// TIA Portal project "Kemence" (V15.1)

(* hardware
DEVICE "HMI_1"  KTP600 Basic color PN
   slot 0: "HMI_1"  KTP600 Basic color PN  6AV6 647-0AD11-3AX0  12.0.0.0
   slot 1: "HMI_RT_1"  KTP600 Basic color PN  6AV6 647-0AD11-3AX0  12.0.0.0
   slot 5: "HMI_1.IE_CP_1"  PROFINET Interface  12.0.0.0
      slot 1: "PROFINET Interface_1"  PROFINET Interface
         slot 1: "Port_1"  Port
DEVICE "S7300/ET200M station_2"  S7-300 station
   slot 0: "Rail_0"  Rail  6ES7 390-1***0-0AA0
   slot 2: "PLC_2"  CPU 314C-2 PN/DP  6ES7 314-6EH04-0AB0  V3.3
      slot 2: "PROFINET interface_1"  PN-IO
         slot 1: "Port_1"  Port
         slot 2: "Port_2"  Port
      slot 5: "DI 24/DO 16_1"  DI24/DO16
      slot 6: "AI 5/AO 2_1"  AI5/AO2
      slot 7: "Count_1"  Counter
      slot 8: "Positioning_1"  Positioning
*)

// ===== PLC "PLC_2"  CPU 314C-2 PN/DP =====

VAR_GLOBAL   // PLC tag table "Default tag table"
   "Homerseklet" AT %IW808 : Int;
   "Ki" AT %Q136.0 : Bool;
   "Orajel" AT %M0.5 : Bool;
END_VAR

DATA_BLOCK "Valtozoim"   // DB1
{ S7_Optimized_Access := 'FALSE' }
VERSION : 0.1
   VAR
      Aktualis : Int;
      Eloirt : Int;
      Hiszterezis : Int;
      Start1 : Bool;
      Start2 : Bool;
      Start3 : Bool;
      "On/Off" : Bool;
      Eloirt_plusz_Hister : Int;
      Eloirt_minus_Hister : Int;
      Kimenet : Bool;
      Komment : Bool;
      Error : Int;
      U : Int;
      Kp : Int;
      Pulse : Bool := true;
   END_VAR
BEGIN
END_DATA_BLOCK

DATA_BLOCK "Harmadik_pont"   // DB5
{ S7_Optimized_Access := 'FALSE' }
VERSION : 0.1
   VAR
      Man_on : Bool;
      PID : Bool;
      CYKLE_TIME : Time;
      Eloirt_REAL : Real;
      Aktualis_REAL : Real;
      Kp_REAL : Real;
      Integralasi_periodus : Time;
      Derivalasi_periodus : Time;
      Felso_hatar : Real;
      Also_hatar : Real;
      szabalyzo_jel : Real;
      Aktualis_DINT : DInt;
      Eloirt_DINT : DInt;
      KP_REAL_1 : Real;
      U_DINT : DInt;
      U_INT : Int;
   END_VAR
BEGIN
END_DATA_BLOCK

FUNCTION "Block_2" : Void   // FC1, LAD
{ S7_Optimized_Access := 'FALSE' }
VERSION : 0.1
BEGIN

REGION Network 1
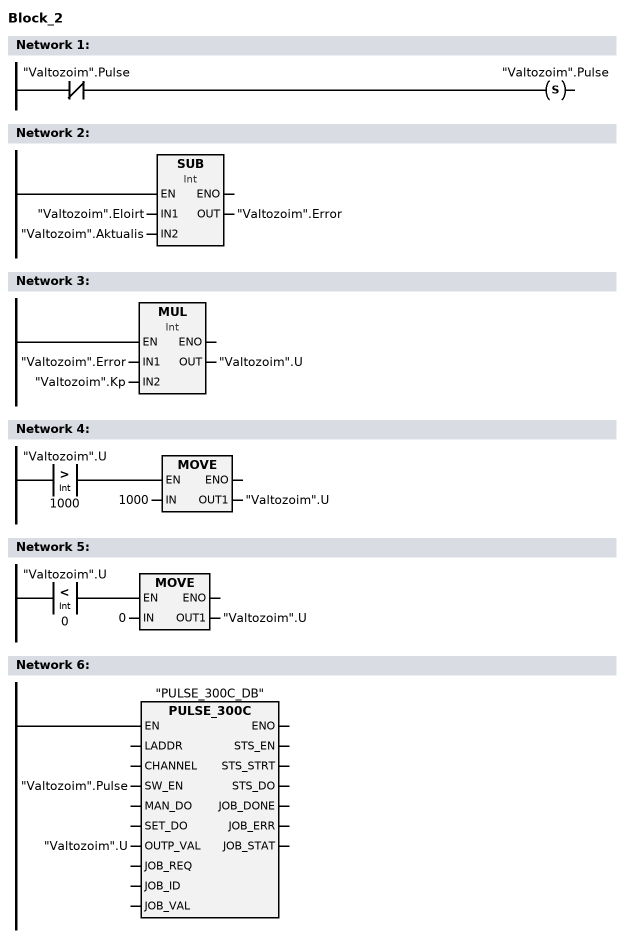
   RUNG wire#powerrail
      I_Contact( "Valtozoim".Pulse )
      S_Coil( "Valtozoim".Pulse )
   END_RUNG
   // the same network as SCL:
   IF NOT "Valtozoim".Pulse THEN "Valtozoim".Pulse := TRUE; END_IF;
END_REGION

REGION Network 2
   RUNG wire#powerrail
      { S7_Templates := "SrcType := Int"; S7_GenerateENO := "TRUE" } Sub(in1 := "Valtozoim".Eloirt, in2 := "Valtozoim".Aktualis, out => "Valtozoim".Error)
   END_RUNG
   // the same network as SCL:
   "Valtozoim".Error := "Valtozoim".Eloirt - "Valtozoim".Aktualis;
END_REGION

REGION Network 3
   RUNG wire#powerrail
      { S7_Templates := "SrcType := Int"; S7_GenerateENO := "TRUE" } Mul(in1 := "Valtozoim".Error, in2 := "Valtozoim".Kp, out => "Valtozoim".U)
   END_RUNG
   // the same network as SCL:
   "Valtozoim".U := "Valtozoim".Error * "Valtozoim".Kp;
END_REGION

REGION Network 4
   RUNG wire#powerrail
      { S7_Templates := "SrcType := Int" } GT_Contact(in1 := "Valtozoim".U, in2 := 1000)
      { S7_GenerateENO := "TRUE" } Move(in := 1000, out1 => "Valtozoim".U)
   END_RUNG
   // the same network as SCL:
   IF "Valtozoim".U > 1000 THEN "Valtozoim".U := 1000; END_IF;
END_REGION

REGION Network 5
   RUNG wire#powerrail
      { S7_Templates := "SrcType := Int" } LT_Contact(in1 := "Valtozoim".U, in2 := 0)
      { S7_GenerateENO := "TRUE" } Move(in := 0, out1 => "Valtozoim".U)
   END_RUNG
   // the same network as SCL:
   IF "Valtozoim".U < 0 THEN "Valtozoim".U := 0; END_IF;
END_REGION

REGION Network 6
   "PULSE_300C_DB"(SW_EN := "Valtozoim".Pulse, OUTP_VAL := "Valtozoim".U);   // PULSE_300C
END_REGION
END_FUNCTION

FUNCTION "Block_1" : Void   // FC2, LAD
{ S7_Optimized_Access := 'FALSE' }
VERSION : 0.1
BEGIN

REGION Network 1
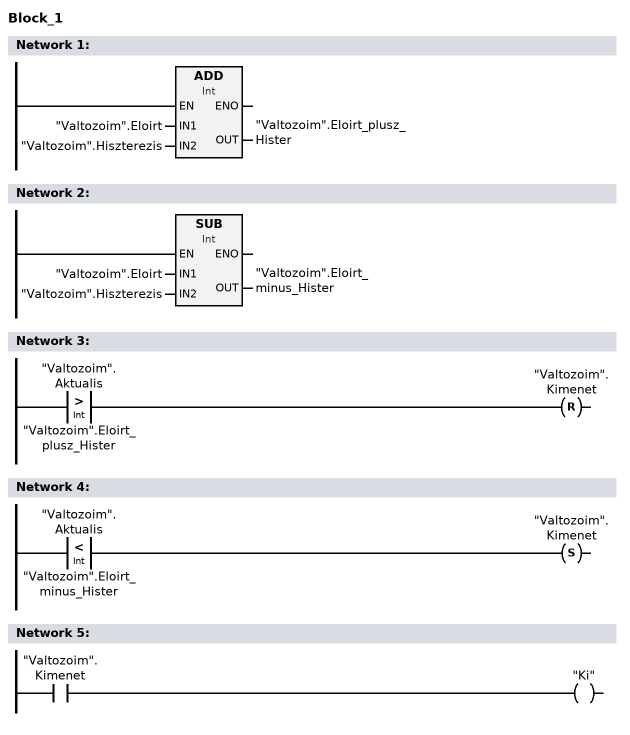
   RUNG wire#powerrail
      { S7_Templates := "SrcType := Int"; S7_GenerateENO := "TRUE" } Add(in1 := "Valtozoim".Eloirt, in2 := "Valtozoim".Hiszterezis, out => "Valtozoim".Eloirt_plusz_Hister)
   END_RUNG
   // the same network as SCL:
   "Valtozoim".Eloirt_plusz_Hister := "Valtozoim".Eloirt + "Valtozoim".Hiszterezis;
END_REGION

REGION Network 2
   RUNG wire#powerrail
      { S7_Templates := "SrcType := Int"; S7_GenerateENO := "TRUE" } Sub(in1 := "Valtozoim".Eloirt, in2 := "Valtozoim".Hiszterezis, out => "Valtozoim".Eloirt_minus_Hister)
   END_RUNG
   // the same network as SCL:
   "Valtozoim".Eloirt_minus_Hister := "Valtozoim".Eloirt - "Valtozoim".Hiszterezis;
END_REGION

REGION Network 3
   RUNG wire#powerrail
      { S7_Templates := "SrcType := Int" } GT_Contact(in1 := "Valtozoim".Aktualis, in2 := "Valtozoim".Eloirt_plusz_Hister)
      R_Coil( "Valtozoim".Kimenet )
   END_RUNG
   // the same network as SCL:
   IF "Valtozoim".Aktualis > "Valtozoim".Eloirt_plusz_Hister THEN "Valtozoim".Kimenet := FALSE; END_IF;
END_REGION

REGION Network 4
   RUNG wire#powerrail
      { S7_Templates := "SrcType := Int" } LT_Contact(in1 := "Valtozoim".Aktualis, in2 := "Valtozoim".Eloirt_minus_Hister)
      S_Coil( "Valtozoim".Kimenet )
   END_RUNG
   // the same network as SCL:
   IF "Valtozoim".Aktualis < "Valtozoim".Eloirt_minus_Hister THEN "Valtozoim".Kimenet := TRUE; END_IF;
END_REGION

REGION Network 5
   RUNG wire#powerrail
      Contact( "Valtozoim".Kimenet )
      Coil( "Ki" )
   END_RUNG
   // the same network as SCL:
   "Ki" := "Valtozoim".Kimenet;
END_REGION
END_FUNCTION

FUNCTION "Block_3" : Void   // FC3, LAD
{ S7_Optimized_Access := 'FALSE' }
VERSION : 0.1
BEGIN

REGION Network 1
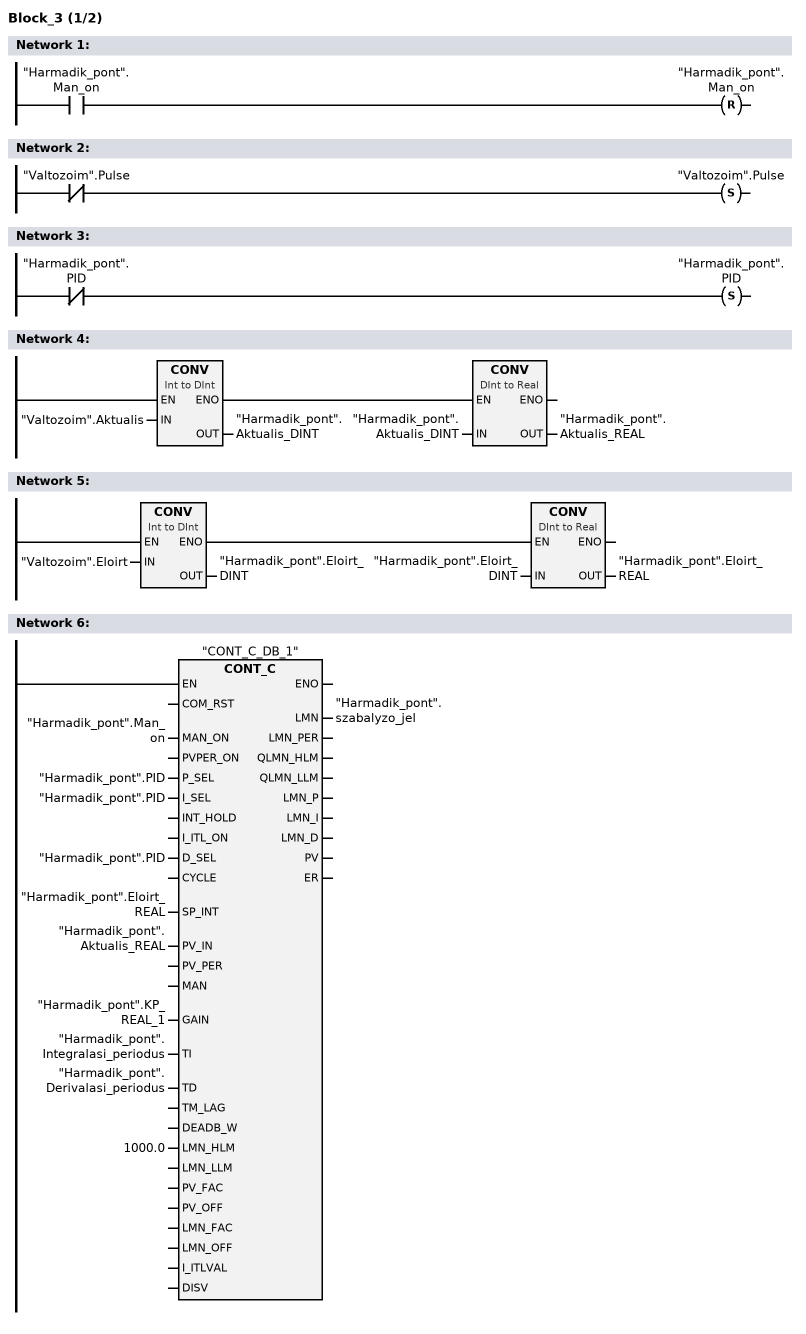
   RUNG wire#powerrail
      Contact( "Harmadik_pont".Man_on )
      R_Coil( "Harmadik_pont".Man_on )
   END_RUNG
   // the same network as SCL:
   IF "Harmadik_pont".Man_on THEN "Harmadik_pont".Man_on := FALSE; END_IF;
END_REGION

REGION Network 2
   RUNG wire#powerrail
      I_Contact( "Valtozoim".Pulse )
      S_Coil( "Valtozoim".Pulse )
   END_RUNG
   // the same network as SCL:
   IF NOT "Valtozoim".Pulse THEN "Valtozoim".Pulse := TRUE; END_IF;
END_REGION

REGION Network 3
   RUNG wire#powerrail
      I_Contact( "Harmadik_pont".PID )
      S_Coil( "Harmadik_pont".PID )
   END_RUNG
   // the same network as SCL:
   IF NOT "Harmadik_pont".PID THEN "Harmadik_pont".PID := TRUE; END_IF;
END_REGION

REGION Network 4
   RUNG wire#powerrail
      { S7_Templates := "[SrcType := Int, DestType := DInt]"; S7_GenerateENO := "TRUE" } Convert(in := "Valtozoim".Aktualis, out => "Harmadik_pont".Aktualis_DINT)
      { S7_Templates := "[SrcType := DInt, DestType := Real]"; S7_GenerateENO := "TRUE" } Convert(in := "Harmadik_pont".Aktualis_DINT, out => "Harmadik_pont".Aktualis_REAL)
   END_RUNG
   // the same network as SCL:
   // ENO of a box is taken as its EN; it also drops when the box reports an error
   "Harmadik_pont".Aktualis_DINT := INT_TO_DINT("Valtozoim".Aktualis);
   "Harmadik_pont".Aktualis_REAL := DINT_TO_REAL("Harmadik_pont".Aktualis_DINT);
END_REGION

REGION Network 5
   RUNG wire#powerrail
      { S7_Templates := "[SrcType := Int, DestType := DInt]"; S7_GenerateENO := "TRUE" } Convert(in := "Valtozoim".Eloirt, out => "Harmadik_pont".Eloirt_DINT)
      { S7_Templates := "[SrcType := DInt, DestType := Real]"; S7_GenerateENO := "TRUE" } Convert(in := "Harmadik_pont".Eloirt_DINT, out => "Harmadik_pont".Eloirt_REAL)
   END_RUNG
   // the same network as SCL:
   // ENO of a box is taken as its EN; it also drops when the box reports an error
   "Harmadik_pont".Eloirt_DINT := INT_TO_DINT("Valtozoim".Eloirt);
   "Harmadik_pont".Eloirt_REAL := DINT_TO_REAL("Harmadik_pont".Eloirt_DINT);
END_REGION

REGION Network 6
   "CONT_C_DB_1"(MAN_ON := "Harmadik_pont".Man_on,   // CONT_C
                 P_SEL := "Harmadik_pont".PID,
                 I_SEL := "Harmadik_pont".PID,
                 D_SEL := "Harmadik_pont".PID,
                 SP_INT := "Harmadik_pont".Eloirt_REAL,
                 PV_IN := "Harmadik_pont".Aktualis_REAL,
                 GAIN := "Harmadik_pont".KP_REAL_1,
                 TI := "Harmadik_pont".Integralasi_periodus,
                 TD := "Harmadik_pont".Derivalasi_periodus,
                 LMN_HLM := 1000.0,
                 LMN => "Harmadik_pont".szabalyzo_jel);
END_REGION

REGION Network 7
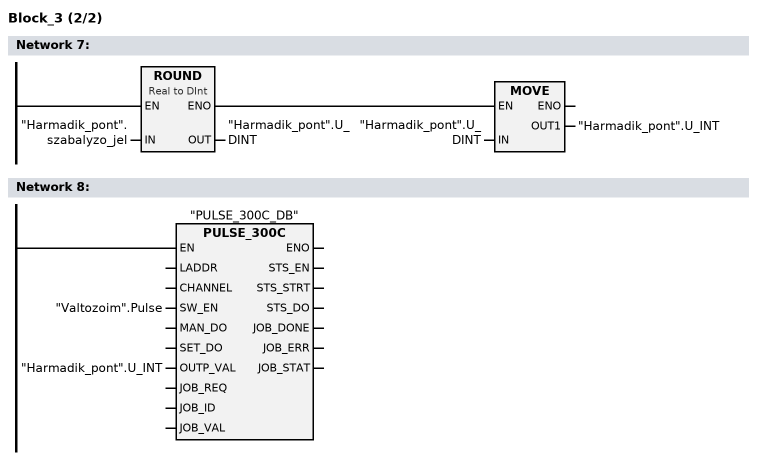
   RUNG wire#powerrail
      { S7_Templates := "[SrcType := Real, DestType := DInt]"; S7_GenerateENO := "TRUE" } Round(in := "Harmadik_pont".szabalyzo_jel, out => "Harmadik_pont".U_DINT)
      { S7_GenerateENO := "TRUE" } Move(in := "Harmadik_pont".U_DINT, out1 => "Harmadik_pont".U_INT)
   END_RUNG
   // the same network as SCL:
   // ENO of a box is taken as its EN; it also drops when the box reports an error
   "Harmadik_pont".U_DINT := ROUND("Harmadik_pont".szabalyzo_jel);
   "Harmadik_pont".U_INT := "Harmadik_pont".U_DINT;
END_REGION

REGION Network 8
   "PULSE_300C_DB"(SW_EN := "Valtozoim".Pulse, OUTP_VAL := "Harmadik_pont".U_INT);   // PULSE_300C
END_REGION
END_FUNCTION

ORGANIZATION_BLOCK "Main"   // OB1, LAD
TITLE = "Main Program Sweep (Cycle)"
{ S7_Optimized_Access := 'FALSE' }
VERSION : 0.1
   VAR_TEMP
      OB1_EV_CLASS : Byte;   // Bits 0-3 = 1 (Coming event), Bits 4-7 = 1 (Event class 1)
      OB1_SCAN_1 : Byte;   // 1 (Cold restart scan 1 of OB 1), 3 (Scan 2-n of OB 1)
      OB1_PRIORITY : Byte;   // Priority of OB Execution
      OB1_OB_NUMBR : Byte;   // 1 (Organization block 1, OB1)
      OB1_RESERVED_1 : Byte;   // Reserved for system
      OB1_RESERVED_2 : Byte;   // Reserved for system
      OB1_PREV_CYCLE : Int;   // Cycle time of previous OB1 scan (milliseconds)
      OB1_MIN_CYCLE : Int;   // Minimum cycle time of OB1 (milliseconds)
      OB1_MAX_CYCLE : Int;   // Maximum cycle time of OB1 (milliseconds)
      OB1_DATE_TIME : Date_And_Time;   // Date and time OB1 started
   END_VAR
BEGIN

REGION Network 1
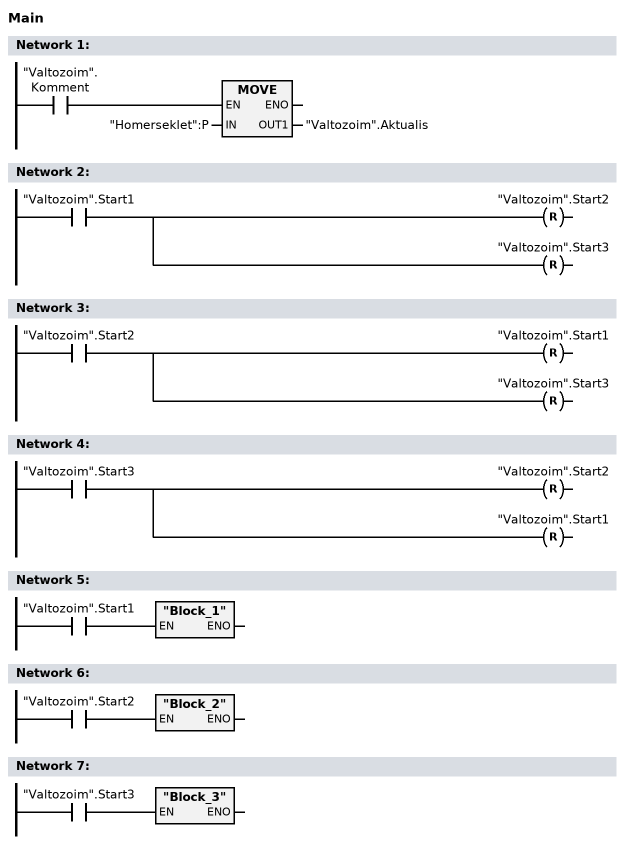
   RUNG wire#powerrail
      Contact( "Valtozoim".Komment )
      { S7_GenerateENO := "TRUE" } Move(in := "Homerseklet":P, out1 => "Valtozoim".Aktualis)
   END_RUNG
   // the same network as SCL:
   IF "Valtozoim".Komment THEN "Valtozoim".Aktualis := "Homerseklet":P; END_IF;
END_REGION

REGION Network 2
   RUNG wire#powerrail
      Contact( "Valtozoim".Start1 )
      wire#w1
      R_Coil( "Valtozoim".Start2 )
   END_RUNG
   RUNG wire#w1
      R_Coil( "Valtozoim".Start3 )
   END_RUNG
   // the same network as SCL:
   IF "Valtozoim".Start1 THEN
       "Valtozoim".Start2 := FALSE;
       "Valtozoim".Start3 := FALSE;
   END_IF;
END_REGION

REGION Network 3
   RUNG wire#powerrail
      Contact( "Valtozoim".Start2 )
      wire#w1
      R_Coil( "Valtozoim".Start1 )
   END_RUNG
   RUNG wire#w1
      R_Coil( "Valtozoim".Start3 )
   END_RUNG
   // the same network as SCL:
   IF "Valtozoim".Start2 THEN
       "Valtozoim".Start1 := FALSE;
       "Valtozoim".Start3 := FALSE;
   END_IF;
END_REGION

REGION Network 4
   RUNG wire#powerrail
      Contact( "Valtozoim".Start3 )
      wire#w1
      R_Coil( "Valtozoim".Start2 )
   END_RUNG
   RUNG wire#w1
      R_Coil( "Valtozoim".Start1 )
   END_RUNG
   // the same network as SCL:
   IF "Valtozoim".Start3 THEN
       "Valtozoim".Start2 := FALSE;
       "Valtozoim".Start1 := FALSE;
   END_IF;
END_REGION

REGION Network 5
   RUNG wire#powerrail
      Contact( "Valtozoim".Start1 )
      "Block_1"()
   END_RUNG
   // the same network as SCL:
   IF "Valtozoim".Start1 THEN "Block_1"(); END_IF;
END_REGION

REGION Network 6
   RUNG wire#powerrail
      Contact( "Valtozoim".Start2 )
      "Block_2"()
   END_RUNG
   // the same network as SCL:
   IF "Valtozoim".Start2 THEN "Block_2"(); END_IF;
END_REGION

REGION Network 7
   RUNG wire#powerrail
      Contact( "Valtozoim".Start3 )
      "Block_3"()
   END_RUNG
   // the same network as SCL:
   IF "Valtozoim".Start3 THEN "Block_3"(); END_IF;
END_REGION
END_ORGANIZATION_BLOCK

(* ===== HMI "HMI_RT_1" =====
system functions are stored by id; their names below are inferred from use
connection "HMI_Connection_1": ETHERNET, SIMATIC S7 300/400 MPI

HMI tags "Default tag table"
   "Valtozoim_Hiszterezis" : Int = PLC Valtozoim.Hiszterezis AT %DB1.DBW4, 100 ms
   "Valtozoim_Aktualis" : Int = PLC Valtozoim.Aktualis AT %DB1.DBW0, 100 ms
   "Valtozoim_Eloirt" : Int = PLC Valtozoim.Eloirt AT %DB1.DBW2, 100 ms
   "Valtozoim_Start1" : Bool = PLC Valtozoim.Start1 AT %DB1.DBX6.0, 100 ms
   "Valtozoim_Start2" : Bool = PLC Valtozoim.Start2 AT %DB1.DBX6.1, 100 ms
   "Valtozoim_Start3" : Bool = PLC Valtozoim.Start3 AT %DB1.DBX6.2, 100 ms
   "Valtozoim_Kimenet" : Bool = PLC Valtozoim.Kimenet AT %DB1.DBX12.0, 100 ms
   "Valtozoim_Kp" : Int = PLC Valtozoim.Kp AT %DB1.DBW18, 1 s
   "Valtozoim_U" : Int = PLC Valtozoim.U AT %DB1.DBW16, 1 s
   "Harmadik_pont_KP_REAL_1" : Real = PLC Harmadik_pont.KP_REAL_1 AT %DB5.DBD46, 1 s
   "Harmadik_pont_Derivalasi_periodus" : Time = PLC Harmadik_pont.Derivalasi_periodus AT %DB5.DBD22, 1 s
   "Harmadik_pont_Integralasi_periodus" : Time = PLC Harmadik_pont.Integralasi_periodus AT %DB5.DBD18, 1 s
   "Harmadik_pont_U_INT" : Int = PLC Harmadik_pont.U_INT AT %DB5.DBW54, 1 s

screen "Root screen" 320x240, template "Template_1"
   TextField "HmiScreenItemData" at 32,34 size 256x44; Text 'Kemence vezérlés'
   Button "Button_1" at 32,94 size 116x31; TextOff 'On/Off kapcsoló'
      on Press: ActivateScreen("Screen_1", 0)
   Button "Button_2" at 176,95 size 119x30; TextOff 'Proporcionális'
      on Press: ActivateScreen("Screen_2", 0)
   Button "Button_3" at 64,144 size 215x33; TextOff 'PID szabályzás'
      on Press: ActivateScreen("Screen_3", 0)

Template "Template_1" 320x240
   Button "Exit" at 266,202 size 52x37; TextOn 'Exit'; TextOff 'Exit'; PictureOn "ExitRuntime_KTP600_Basic_color_PN"; PictureOff "ExitRuntime_KTP600_Basic_color_PN"
      on Release: StopRuntime(0)
   Button "Template_Button" at 213,202 size 52x37; TextOff 'Text'
   Button "Template_Button_1" at 160,202 size 52x37; TextOff 'Text'
   Button "Template_Button_2" at 107,202 size 52x37; TextOff 'Text'
   Button "Start screen" at 54,202 size 52x37; TextOn 'Start screen'; TextOff 'Start screen'; PictureOn "NavigateHome_KTP600_Basic_color_PN"; PictureOff "NavigateHome_KTP600_Basic_color_PN"
      on Release: ActivateScreen("Root screen", 0)
   Button "Alarms" at 1,202 size 52x37; TextOn 'Alarms'; TextOff 'Alarms'; PictureOn "AlarmDisplay_KTP600_Basic_color_PN"; PictureOff "AlarmDisplay_KTP600_Basic_color_PN"
      on Release: function_ef3f5d25("Alarm window_Unacknowledged", -1)
   DateTimeField "HmiScreenItemData" at 235,19 size 85x19
   DateTimeField "HmiScreenItemData_1" at 235,0 size 85x19
   GraphicView "Logo" at 0,0 size 67x38; Picture "Logo of HMI_1"

screen "Screen_1" 320x240
   TextField "HmiScreenItemData" at 42,7 size 256x44; Text 'Kemence vezérlés'
   TextField "HmiScreenItemData_1" at 8,80 size 108x29; Text 'Előírt hőmérséklet:'
   TextField "HmiScreenItemData_2" at 3,105 size 120x25; Text 'Aktuális hőmérséklet:'
   IOField "I/O field_1" at 124,111 size 54x18; FormatPattern s99999
      ProcessValue <- "Valtozoim_Aktualis"
   IOField "I/O field_2" at 124,82 size 96x23; FormatPattern s99999
      ProcessValue <- "Valtozoim_Eloirt"
   Button "Button_1" at 104,158 size 96x32; TextOff 'Start'
      on Press: SetBit("Valtozoim_Start1")
   Button "Button_2" at 114,198 size 76x25; TextOff 'Home'
      on Press: ActivateScreen("Root screen", 0); ResetBit("Valtozoim_Start1"); ResetBit("Valtozoim_Start2"); ResetBit("Valtozoim_Start3"); ResetBit("Valtozoim_Kimenet")
   Circle "Circle_1" at 232,147 size 25x25
      Appearance <- "Valtozoim_Kimenet"
   TextField "HmiScreenItemData_3" at 213,121 size 72x29; Text 'Q136.0'
   TextField "HmiScreenItemData_5" at 39,30 size 256x44; Text 'On/Off kapcsoló'
   TextField "HmiScreenItemData_6" at 9,131 size 96x24; Text 'Hiszterézis:'
   IOField "I/O field_3" at 124,135 size 43x20; FormatPattern s99
      ProcessValue <- "Valtozoim_Hiszterezis"

screen "Screen_2" 320x240
   TextField "HmiScreenItemData" at 42,7 size 256x44; Text 'Text'
   TextField "HmiScreenItemData_1" at 5,70 size 120x44; Text 'Előírt hőmérséklet:'
   TextField "HmiScreenItemData_2" at 5,96 size 120x44; Text 'Aktuális hőmérséklet:'
   IOField "I/O field_1" at 124,111 size 44x18; FormatPattern s99999
      ProcessValue <- "Valtozoim_Aktualis"
   IOField "I/O field_2" at 124,82 size 96x23; FormatPattern s99999
      ProcessValue <- "Valtozoim_Eloirt"
   Button "Button_1" at 104,158 size 96x32; TextOff 'Start'
      on Press: SetBit("Valtozoim_Start2")
   Button "Button_2" at 114,198 size 76x25; TextOff 'Home'
      on Press: ActivateScreen("Root screen", 0); ResetBit("Valtozoim_Start1"); ResetBit("Valtozoim_Start2"); ResetBit("Valtozoim_Start3")
   TextField "HmiScreenItemData_5" at 37,2 size 256x44; Text 'Proporcionális szabályzás'
   TextField "HmiScreenItemData_6" at 9,120 size 120x44; Text 'Hangolási tényező:'
   IOField "I/O field_3" at 124,135 size 43x20; FormatPattern s99
      ProcessValue <- "Valtozoim_Kp"
   Bar "Bar_1" at 236,72 size 80x146; MinimumValue 0; MaximumValue 1000
      ProcessValue <- "Valtozoim_U"

screen "Screen_3" 320x240
   TextField "HmiScreenItemData" at 42,-9 size 256x44; Text 'Text'
   TextField "HmiScreenItemData_1" at 5,58 size 120x17; Text 'Előírt hőmérséklet:'
   TextField "HmiScreenItemData_2" at 5,85 size 120x17; Text 'Aktuális hőmérséklet:'
   IOField "I/O field_1" at 124,84 size 50x18; FormatPattern s99999
      ProcessValue <- "Valtozoim_Aktualis"
   IOField "I/O field_2" at 124,57 size 96x23; FormatPattern s99999
      ProcessValue <- "Valtozoim_Eloirt"
   Button "Button_1" at 116,175 size 96x32; TextOff 'Start'
      on Press: SetBit("Valtozoim_Start3")
   Button "Button_2" at 127,210 size 76x25; TextOff 'Home'
      on Press: ActivateScreen("Root screen", 0); ResetBit("Valtozoim_Start1"); ResetBit("Valtozoim_Start2"); ResetBit("Valtozoim_Start3")
   TextField "HmiScreenItemData_5" at 36,0 size 256x44; Text 'PID szabályzás'
   TextField "HmiScreenItemData_6" at 10,111 size 21x25; Text 'Kp'
   IOField "I/O field_3" at 36,116 size 50x20; FormatPattern s999999999.999
      ProcessValue <- "Harmadik_pont_KP_REAL_1"
   Bar "Bar_1" at 236,72 size 80x146; MinimumValue 0; MaximumValue 1000
      ProcessValue <- "Harmadik_pont_U_INT"
   TextField "HmiScreenItemData_3" at 3,175 size 34x25; Text 'TI'
   IOField "I/O field_4" at 36,179 size 50x20; FormatPattern s9999999999
      ProcessValue <- "Harmadik_pont_Integralasi_periodus"
   TextField "HmiScreenItemData_4" at 5,145 size 28x25; Text 'TD'
   IOField "I/O field_5" at 36,148 size 50x20; FormatPattern s9999999999
      ProcessValue <- "Harmadik_pont_Derivalasi_periodus"
   TextField "HmiScreenItemData_7" at 91,110 size 21x25; Text 'ms'
   TextField "HmiScreenItemData_8" at 92,143 size 21x25; Text 'ms'
   TextField "HmiScreenItemData_9" at 92,176 size 21x25; Text 'ms'
*)